# B&R Automation Studio project TD52 (part 146)

#### Stat_Obj.st - Cyclic code
```iecst
(*******************************************************************************
AGGR: read and write start statistic to windows file system	(cyclic)

This code is confidential and proprietary to the INNIO Company.
It may not be used in any form, or reproduced in any manner, without the express
written permission of the INNIO Company.
Copyright, INNIO Company, 2025

Customized modifications: -
------------------------

History:
-------
V4.06.00 	13-03-2018 	502423184	generated out of Stat_File
V4.06.01	20-07-2018	502423184	Erweitert um: LastRunInfo, TiAuxRel, Update(skip data info)
V4.12.00	29-03-2023	Kafka,		CBM HMI Handshake for Statistic Files
V4.13.0		30-10-2023	Kafka,		solve special sign issue
V4.14.0		27-02-2025	Perktold	added Ti_Purge_Dur to start statistic (new strVersion 4.14.0)

Instructions for use:
--------------------
Update Version number in the INIT program part and in history above!
Always increase the Version Number +0.00.01, if changes are made.

100ms+ Task class (TC6)

Outstandings:
------------
*******************************************************************************)

PROGRAM _INIT
(** A: Version Number *)
	strVersion			:=	'4.14.00';				(* Always increase the Version Number +0.00.01, if changes are made. *)

(** B: Initialize variables *)
	bOK 			:=	FALSE;
	aData			:=	ADR(szData);
	aTemp			:=	ADR(strTemp);
	lines			:=	1;
	strcpy(ADR(ModulName),ADR('CBM::Statistic'));

	pm_len			:=	SIZEOF(DerString_Stat);		(* define data length of permenent memory				*)

	DatObjInfo_01.enable		:=	TRUE;
	DatObjInfo_01.pName			:=	ADR(ModulName);

	DatObjCreate_01.enable		:=	TRUE;			(* enable create permanent memory data module FUB 		*)
	DatObjCreate_01.grp			:=	0;				(* must to be set to zero                  				*)
	DatObjCreate_01.pName		:=	ADR(ModulName);	(* set permanent memory data module name             	*)
	DatObjCreate_01.len			:=	pm_len;			(* set length of permanent memory data module         	*)
	DatObjCreate_01.MemType		:=	doUSRROM;		(* create permanent memory data module at USERROM   	*)
	DatObjCreate_01.Option		:=	0;				(* cyclic checksum monitoring is on            			*)
	DatObjCreate_01.pCpyData	:=	0;				(* no data will be copied do the perm. mem. data module	*)

	DatObjWrite_01.enable		:=	TRUE;			(* enable permanent memory data module read FUB 		*)
	DatObjWrite_01.Offset		:=	0;				(* start at memory offest zero                  		*)
	DatObjWrite_01.pSource		:=	ADR(DerString_Stat);	(* set permanent memory data module name		*)
	DatObjWrite_01.len			:=	pm_len;			(* set length ofpermanent memory data module        	*)

(** C: Functionality test and validation *)
	TON_Test.PT		:=	T#1m;
	bTest_Ena		:=	FALSE;

END_PROGRAM

PROGRAM _CYCLIC

(** 0: Functionality test and validation *)
	IF bTest_Ena THEN
		TON_Test.IN := NOT TON_Test.Q;
		TON_Test();

		IF TON_Test.Q THEN
			bStat_Write := TRUE;
			test_cnt	:=	(1 + test_cnt) MOD 3;
			iStat_Mode	:=	1 + test_cnt;
			CASE iStat_Mode OF
				1,2: 	lines			:=	StatSize;
				3:		lines			:=	Err.Size;
			END_CASE
		END_IF
	END_IF

(** 1: Triggers *)

(** 1.1: Statistic Triggers: manual trigger / automatic trigger every 100 starts *)
	IF iStep = _IDLE THEN
		IF VIS2MM.Stat.bTrig THEN
			bStat_Write		:=	TRUE;
			iStat_Mode		:=	MAN;
			lines			:=	StatSize;
		END_IF
		IF bStat_Trigger THEN
			bStat_Write		:=	TRUE;
			iStat_Mode		:=	AUTO;
			lines			:=	StatSize;
		END_IF
		VIS2MM.Stat.bTrig	:=	FALSE;
		bStat_Trigger		:=	FALSE;
	END_IF

(** 1.2: daily trigger for error counter myPlant *)
	IF NOT IN_CB.tPB2MM.bParaSetupOk THEN
		day_old			:=	tRealTime.day;
	END_IF
	IF tRealTime.day <> day_old THEN
		day_old			:=	tRealTime.day;
		bDaily_Trigger	:=	Para.iDailyTrigger_Ena > 0;
	END_IF

(** 1.3: Error Counter Trigger *)
	IF Para.bSA_PBC_Active AND iStep = _IDLE THEN
		IF VIS2MM.ErrCnt.bTrig OR bDaily_Trigger THEN
			bStat_Write		:=	TRUE;
			iStat_Mode		:=	ERRCNT;
			lines			:=	Err.Size;
		END_IF
		VIS2MM.ErrCnt.bTrig	:=	FALSE;
		bDaily_Trigger		:=	FALSE;
	END_IF

(** 2: initialiate file write *)
IF EDGEPOS(bStat_Write) THEN
	iStep 		:=	_BEGIN;
	bWrite		:=	TRUE;
	iZeile		:=	0;
	iOffset		:=	0;
	strFile			:=	'';																			(* create filename *)
	WRITE_Date(ADR(strFile),tRealTime);																(* Date *)
	IF iStat_Mode = ERRCNT THEN		strcat(ADR(strFile), ADR('_ErrCnt'));							(* _Name *)
	ELSE							strcat(ADR(strFile), ADR('_Statistic'));	END_IF
	strcat(ADR(strFile), ADR('_'));	strcat(ADR(strFile), ADR(IN_CB.szOrderID));						(* _OrderID *)
	strcat(ADR(strFile), ADR('_'));	itoa(IN_CB.iEngID, 	 aTemp);	strcat(ADR(strFile), aTemp);	(* _EngineID *)
	IF iStat_Mode = AUTO THEN		strcat(ADR(strFile), ADR('_Auto'));								(* _Mode *)
	ELSIF iStat_Mode = MAN THEN		strcat(ADR(strFile), ADR('_Man'));			END_IF
	strcat(ADR(strFile), ADR('.csv'));																(* .csv *)
END_IF

(** 3: when write process is done then reset event bit *)
	IF EDGENEG(bWrite) THEN
		bStat_Write	:=	FALSE;
	END_IF

(** 4: State machine *)
	CASE iStep OF
(** 4.1: write filename and version *)
	_BEGIN:
		szData		:=	'';
		strcat(aData, ADR('<STATS_NAME>'));																						(* ------------ *)
		strcat(aData, ADR(strFile));																							(* file name *)
		strcat(aData, ADR('</STATS_NAME><STATS_FILE>'));																		(* ------------ *)
		strcat(aData, ADR(strGEProp));																							(* GE prop info *)
		strcat(aData, ADR(strLine));																							(* ------------ *)
		strcat(aData, ADR('File_Version;'));	WRITE_STRING(ADR(strVersion),aData);				strcat(aData, ADR('$n'));	(* File version *)
		strcat(aData, ADR('Creation_Date;'));	WRITE_TS(tTimeStamp, aData);						strcat(aData, ADR('$n'));	(* Date & Time *)
		strcat(aData, ADR('J_Number;'));		WRITE_STRING(ADR(IN_CB.szOrderID),aData);			strcat(aData, ADR('$n'));	(* J Number *)
		strcat(aData, ADR('Motor_Number;'));	WRITE_DINT(IN_CB.iEngID,aData);						strcat(aData, ADR('$n'));	(* Serial ID *)
		strcat(aData, ADR('Engine_Type;'));		WRITE_DINT(xEngType.Motortype,aData);				strcat(aData, ADR('$n'));	(* Engine Type *)
		strcat(aData, ADR('Engine_Version;'));	WRITE_STRING(ADR(IN_CB.szEng_Motorversion),aData);	strcat(aData, ADR('$n'));	(* Engine Version *)
		strcat(aData, ADR('Trigger_Event;'));	WRITE_DINT(iStat_Mode,aData);						strcat(aData, ADR('$n'));	(* Trigger *)
		strcat(aData, ADR(strLine));																							(* ------------ *)

		DerString_Stat := '';
		iStrSize	:=	SIZEOF(DerString_Stat);
		iPointer	:=	ADR(DerString_Stat);
		iPointer	:=	save_strcat(ADR(DerString_Stat), iStrSize, iPointer, aData);					(* write data line *)
		iStep		:=	_HEAD;																			(* next step *)

(** 4.2: write file header *)
	_HEAD:
		szData		:=	'';
		IF iStat_Mode = AUTO OR iStat_Mode = MAN THEN													(* Statistic Header *)
			FOR i:=0 TO Stat.iSize DO	IF NOT Stat.i[i].Skip THEN	WRITE_STRING(ADR(Stat.i[i].Name), aData);	END_IF	END_FOR	(* Integer Names *)
			FOR i:=0 TO Stat.sSize DO	IF NOT Stat.s[i].Skip THEN	WRITE_STRING(ADR(Stat.s[i].Name), aData);	END_IF	END_FOR	(* String Names *)
			FOR i:=0 TO Stat.bSize DO	IF NOT Stat.b[i].Skip THEN	WRITE_STRING(ADR(Stat.b[i].Name), aData);	END_IF	END_FOR	(* Boolean Names *)
			FOR i:=0 TO Stat.rSize DO	IF NOT Stat.r[i].Skip THEN	WRITE_STRING(ADR(Stat.r[i].Name), aData);	END_IF	END_FOR	(* Real Names *)
			strcat(aData, ADR('$n'));
			FOR i:=0 TO Stat.iSize DO	IF NOT Stat.i[i].Skip THEN	WRITE_STRING(ADR(Stat.i[i].Unit), aData);	END_IF	END_FOR	(* Integer Units *)
			FOR i:=0 TO Stat.sSize DO	IF NOT Stat.s[i].Skip THEN	strcat(aData, ADR(';'));					END_IF	END_FOR	(* no Units *)
			FOR i:=0 TO Stat.bSize DO	IF NOT Stat.b[i].Skip THEN	strcat(aData, ADR(';'));					END_IF	END_FOR	(* no Units *)
			FOR i:=0 TO Stat.rSize DO	IF NOT Stat.r[i].Skip THEN	WRITE_STRING(ADR(Stat.r[i].Unit), aData);	END_IF	END_FOR	(* Real Units *)
			strcat(aData, ADR('$n'));
		ELSIF iStat_Mode = ERRCNT THEN																	(* ErrCounter Header *)
			strcat(aData, ADR('Reset date; '));			WRITE_TS(Err.tTS_Reset, aData);
			strcat(aData, ADR('$nReset OpHours; '));	itoa(Err.iCnt_OH_Reset,aTemp);	strcat(aData, aTemp);
			strcat(aData, ADR('$nWrite date; '));		WRITE_TS(tTimeStamp, aData);
			strcat(aData, ADR('$nWrite OpHours; '));	itoa(IN_CB.iCnt_OpHours,aTemp);	strcat(aData, aTemp);
			strcat(aData, ADR('$nErrorBit / Measurement; '));
			strcat(aData, ADR('Cyl / SAFI; '));
			strcat(aData, ADR('Counter; '));
			strcat(aData, ADR('First date; '));
			strcat(aData, ADR('Last date; '));
			strcat(aData, ADR('$n'));
		END_IF
		iPointer	:=	save_strcat(ADR(DerString_Stat), iStrSize, iPointer, aData);					(* write data line *)
		iStep		:=	_DATA;																			(* next step *)

(** 4.3: create data lines *)
	_DATA:
		szData		:=	'';																				(* clear previous data *)
		IF iStat_Mode = AUTO OR iStat_Mode = MAN THEN													(* Statistic Data *)
			iIdx	:=	(USINT_TO_INT(Stat.iIdx) - UDINT_TO_INT(iZeile) + USINT_TO_INT(StatSize + 1))MOD (StatSize + 1); (* calculate ring buffer index *)
			FOR i:=0 TO Stat.iSize DO	IF NOT Stat.i[i].Skip THEN	WRITE_DINT(Stat.i[i].Data[iIdx], 					aData);	END_IF	END_FOR
			FOR i:=0 TO Stat.sSize DO	IF NOT Stat.s[i].Skip THEN	WRITE_STRING(ADR(Stat.s[i].Data[iIdx].str), 		aData);	END_IF	END_FOR
			FOR i:=0 TO Stat.bSize DO	IF NOT Stat.b[i].Skip THEN	WRITE_BIT(Stat.b[i].Data[iIdx],						aData);	END_IF	END_FOR
			FOR i:=0 TO Stat.rSize DO	IF NOT Stat.r[i].Skip THEN	WRITE_REAL(Stat.r[i].Data[iIdx], Stat.r[i].Deci,	aData);	END_IF	END_FOR
		ELSIF iStat_Mode = ERRCNT THEN																	(* ErrCounter Data *)
			WRITE_STRING(ADR(ErrName[Err.xErr[iZeile].Name].str), 	aData);
			WRITE_DINT(Err.xErr[iZeile].iNum_Cyl, 					aData);
			WRITE_DINT(UDINT_TO_DINT(Err.xErr[iZeile].iCnt), 		aData);
			WRITE_TS(Err.xErr[iZeile].tTS_First,					aData);
			WRITE_TS(Err.xErr[iZeile].tTS_Last,						aData);
		END_IF
		strcat(aData, ADR('$n'));																		(* Line End *)
		iPointer	:=	save_strcat(ADR(DerString_Stat), iStrSize, iPointer, aData);					(* write data line *)
		IF iZeile < lines THEN			iZeile		:=	MIN(iZeile + 1, lines);							(* next line *)
		ELSE							iStep		:=	_FOOT;											(* next step *)
		END_IF

(** 4.4: create file footer *)
	_FOOT:
		iPointer	:=	save_strcat(ADR(DerString_Stat), iStrSize, iPointer, ADR('END OF FILE $n'));	(* last line *)
		iPointer	:=	save_strcat(ADR(DerString_Stat), iStrSize, iPointer, ADR('</STATS_FILE>'));		(* file end *)
		bWrite		:=	FALSE;																			(* write end *)
		iStep		:=	_EXIST;																			(* next step *)

(** 4.5: check for existing permanent memory data module *)
	_EXIST:
		DatObjInfo_01();
		CASE  DatObjInfo_01.status OF
		_BUSY: 	iStep;																					(* waiting *)
		_OKAY:	iStep 			:= _WRITE;																(* next step --> write the content to the flash disk	*)
				DatObjWrite_01.ident   	:= DatObjInfo_01.ident;											(* set identifier of permanent memory data module		*)
				DatObjWrite_01.len		:= pm_len;
		_DONF:	iStep		:=	_CREATE;																(* next step --> create permanent memory data module	*)
		ELSE	iErrorStep	:=	iStep;
				iStep		:=	_ERROR;
				iError		:=	DatObjInfo_01.status;
		END_CASE

(** 4.6: create permanent memory data module *)
	_CREATE:
		DatObjCreate_01();
		CASE  DatObjCreate_01.status OF
		_BUSY:	iStep;																					(* repeat until generation of permanent memory data module is ready *)
		_OKAY:	DatObjWrite_01.ident   	:= DatObjCreate_01.ident;										(* set identifier of permanent memory data module     	*)
				DatObjWrite_01.len		:= pm_len;
				iStep		:=	_WRITE;																	(* next step --> write the content to the flash disk	*)
		ELSE	iErrorStep	:=	iStep;
				iStep		:=	_ERROR;
				iError		:=	DatObjCreate_01.status;
		END_CASE

(** 4.7: write the content to the flash disk *)
	_WRITE:
		DatObjWrite_01();
	 	CASE DatObjWrite_01.status OF
		_BUSY:	iStep;																					(* repeat until write process of permanent memory data module is done *)
	   	_OKAY:	iStep				:=	_HMI;															(* next step --> wait for HMI to fetch file	*)
				xTON_HMI_Delay.IN	:=	TRUE;
		ELSE	iErrorStep			:=	iStep;
				iStep				:=	_ERROR;
				iError				:=	DatObjWrite_01.status;
		END_CASE

(** 4.8: wait FOR HMI TO fetch file	*)
	_HMI:
		MM2VIS.bStat_isCreated	:= TRUE;
		IF xTON_HMI_Delay.Q OR VIS2MM.bStat_isRead THEN
			iStep				:=	_DONE;																(* next step *)
			xTON_HMI_Delay.IN	:=	FALSE;
			MM2VIS.bStat_isCreated	:=	FALSE;
			VIS2MM.bStat_isRead		:=	FALSE;
		END_IF

(** 4.9: done, go to idle mode	*)
	_DONE:	iStep		:=	_IDLE;

(** 4.10: idle, reset lines	*)
	_IDLE:	iZeile		:=	0;
			iErrorStep	:=	0;

(** 4.11: error step, wait for cold start *)
	_ERROR: iStep;

(** 4.12: catch unexpected states *)
	ELSE	iErrorStep	:=	iStep;
			iStep		:=	_ERROR;
	END_CASE

(** 5: HMI Delay and out interfaces *)
	xTON_HMI_Delay.PT	:=	tiHMI_Delay;
	xTON_HMI_Delay();

	IF xTON_HMI_Delay.PT <> T#0s THEN
		rHMI_Delay	:=	LIMIT(0.0, TIME_TO_REAL(xTON_HMI_Delay.ET) / TIME_TO_REAL(xTON_HMI_Delay.PT), 1.0);
	ELSE
		rHMI_Delay	:=	0;
	END_IF

	IF iStep = _DONE THEN
		MM2VIS.Stat.rSave	:=	1.0;
	ELSIF iStep <> _HMI AND lines <> 0 THEN
		MM2VIS.Stat.rSave	:=	0.5 * UDINT_TO_REAL(iZeile)/UINT_TO_REAL(lines);
	ELSIF iStep = _HMI AND lines <> 0 THEN
		MM2VIS.Stat.rSave	:=	0.5 + 0.5 * rHMI_Delay;
	ELSIF iStep = _HMI AND lines = 0 THEN
		MM2VIS.Stat.rSave	:=	rHMI_Delay;
	END_IF

	MM2VIS.ErrCnt.rSave			:=	MM2VIS.Stat.rSave;

	MM2VIS.Stat.bSave			:=	iStep <> _IDLE AND lines = StatSize;
	MM2VIS.ErrCnt.bSave			:=	iStep <> _IDLE AND lines = Err.Size;

	IF iStep = _IDLE THEN
		MM2VIS.Stat.iStep			:=	USINT_TO_INT(_RDY);
		MM2VIS.ErrCnt.iStep			:=	USINT_TO_INT(_RDY);
	ELSE
		MM2VIS.Stat.iStep			:=	USINT_TO_INT(iStep) * BOOL_TO_INT(lines = StatSize) + _LOCK * BOOL_TO_INT(lines <> StatSize);
		MM2VIS.ErrCnt.iStep			:=	USINT_TO_INT(iStep) * BOOL_TO_INT(lines = Err.Size) + _LOCK * BOOL_TO_INT(lines <> Err.Size);
	END_IF

	MM2VIS.Stat.bLock			:=	iStep <> _IDLE;
	MM2VIS.ErrCnt.bLock			:=	iStep <> _IDLE;

END_PROGRAM
```

#### Stat_Obj.var - Local variables
```iecst
(********************************************************************
 * COPYRIGHT -- INNIO Company
 ********************************************************************
 * Program: PBC_MFile
 * File: PBC_MFile.var
 * Author: 502293141
 * Created: October 23, 2014
 ********************************************************************
 * Local variables of program PBC_MFile
 ********************************************************************)
VAR
	bOK : BOOL;
	strFile : STRING[50];
	iZeile : UDINT;
	iOffset : UDINT;
	iIdx : INT;
	bWrite : BOOL;
	szData : STRING[15000];
	iError : UINT;
	bStat_Write : BOOL;
	iStat_Mode : USINT;
	ModulName : STRING[32];
	pm_len : UDINT := 0;
	day_old : USINT;
	bDaily_Trigger : BOOL := 0;
	iStep : USINT := 0;
	DerString_Stat : STRING[200000];
	iErrorStep : INT;
	TON_Test : TON;
	i : UINT;
	strTemp : STRING[10];
	lines : UINT;
	DatObjCreate_01 : DatObjCreate;
	DatObjWrite_01 : DatObjWrite;
	DatObjInfo_01 : DatObjInfo;
	test_cnt : USINT;
	xTON_HMI_Delay : TON;
	strVersion : STRING[30];
	rHMI_Delay : REAL;
aData : UDINT;
aTemp : UDINT;
iStrSize : UDINT;
iPointer : UDINT;
END_VAR
VAR CONSTANT
	MAN : USINT := 1;
	AUTO : USINT := 2;
	ERRCNT : USINT := 3;
END_VAR
VAR
	bTest_Ena : BOOL := 0;
END_VAR
```

### Program Logical/CBM/Statistic/ErrCnt (IEC, version 4.06.1) - + counts errors

- ErrCnt.st (not readable text: treated as protected, skipped)

#### ErrCnt.var - Local variables
```iecst
(********************************************************************
 * COPYRIGHT -- INNIO Company
 ********************************************************************
 * Program: ErrCnt
 * File: ErrCnt.var
 * Author: 502423184
 * Created: December 14, 2015
 ********************************************************************
 * Local variables of program ErrCnt
 ********************************************************************)
VAR
	iNum_Cyl : USINT;
	iCnt : UINT;
	iCnt_Err : UINT;
	xTON_ErrCnt_Ena : TON;
END_VAR
VAR CONSTANT
	Knock_Int : USINT := 1;
	Knock_Lim : USINT := 2;
	Knock_Lim_Filt : USINT := 3;
	Misf_I : USINT := 4;
	Misf_II : USINT := 5;
	GlowIgn : USINT := 6;
	SensErr : USINT := 7;
	SensFailure : USINT := 8;
	MemBurst : USINT := 9;
	CPSSat : USINT := 0; (*Cylinder pressure sensor saturation - error counter*)
	CompLineCheck : USINT := 10;
	NegPresCheck : USINT := 11;
	PresSlopeCheck : USINT := 12;
	SlowDriftCheck : USINT := 13;
	PmaxLimReached : USINT := 14;
	NegVoltCheck : USINT := 15;
	ConfNotOK : USINT := 16;
	InvalidPar : USINT := 17;
	LimpHome : USINT := 18;
	OptiFreeze : USINT := 19;
END_VAR
```

### Program Logical/CBM/VisCBM (IEC) - Program

#### VisCBM.st - Cyclic code
```iecst
(*******************************************************************************
AGGR: VIS

This code is confidential AND proprietary to the INNIO Company.
It may NOT be used in any form, or reproduced in any manner, without the express
written permission of the INNIO Company.
Copyright, INNIO Company, 2019

Customized modifications: -
------------------------
History:
-------
V4.06.01 	30-07-2018 	502423184		header added, moved rCA_MFBxx to IN_CBM task

Instructions FOR use:
--------------------
- use in a 100ms cycle time

Outstandings:
------------
-

*******************************************************************************)
PROGRAM _INIT

	PINK;
END_PROGRAM

PROGRAM _CYCLIC

(** 1: colormap for that *)
	FOR i:= 1 TO 24 DO
		IF IN_CB.bTripCyl[i]				THEN	MM2VIS.iIdx_CylColor[i]	:=	RED;
		ELSIF IN_CB.bLimpHomeCylRKS_TC5[i]	THEN	MM2VIS.iIdx_CylColor[i]	:=	BLUE;
		ELSIF IN_CB.bLimpHomeCyl[i]			THEN	MM2VIS.iIdx_CylColor[i]	:=	YELLOW;
		ELSIF IN_CB.bSkipCylAct[i]			THEN	MM2VIS.iIdx_CylColor[i]	:=	GREY;
		ELSIF bATDCyl[i]					THEN	MM2VIS.iIdx_CylColor[i]	:=	VIOLET;
		ELSE 						 	 			MM2VIS.iIdx_CylColor[i]	:=	GREEN;
		END_IF
	END_FOR

(** 2: Statistic and CBM Screen visibility **)
	MM2VIS.bScreen_Stat :=	xEngType.Type9 OR Para.bSStat_Ena;
	MM2VIS.bScreen_CBM	:=	xEngType.Type9 OR Para.bSStat_Ena OR Para.bTCBMem_Ena OR Para.bECBMem_Ena OR Para.bSA_PBC_Active;

	MM2VIS.Stat.bScreen		:=	Para.bSStat_Ena;
	MM2VIS.ErrCnt.bScreen	:=	Para.bSA_PBC_Active;
	MM2VIS.TCB.bScreen		:=	Para.bTCBMem_Ena;
	MM2VIS.ECB.bScreen		:=	Para.bECBMem_Ena;

	MM2VIS.bFrictIMEP_Condition_On	:= OUT_CB.bFrictIMEP_Condition_On;

(** 3: SAFI data to HMI *)
	MM2VIS.rCA_MFB10 :=	rCA_MFB10;
	MM2VIS.rCA_MFB90 :=	rCA_MFB90;

END_PROGRAM
```

#### VisCBM.var - Local variables
```iecst
(********************************************************************
 * COPYRIGHT -- INNIO Company
 ********************************************************************
 * Program: VisCBM
 * File: VisCBM.var
 * Author: 105026853
 * Created: January 27, 2016
 ********************************************************************
 * Local variables of program VisCBM
 ********************************************************************)
VAR
	i : USINT;
END_VAR
```

### Program Logical/CBM/GnrlCBM (IEC) - Program

#### GnrlCBM.st - Cyclic code
```iecst
(*******************************************************************************
CBM: general monotioring task  (cyclic)

This code is confidential AND proprietary to the INNIO Company.
It may NOT be used in any form, or reproduced in any manner, without the express
written permission of the INNIO Company.
Copyright, INNIO Company, 2023

- GEN2diag checks the lambda movement AND shut down the engine in CASE OF a friciton event
- FricIMEP checks the friction power AND shut down the engine in CASE OF an increase

Customized modifications: -
------------------------

History:
-------

V4.05.0 xx-xx-2018 	Waldhart, 	created
V4.06.0 24-07-2018 	Waldhart, 	GEN2diag V0.3.9 implemented
		30-07-2018	502423184	replaced Para.bGEN2_preM_Act
V4.07.0 20-09-2018 	Waldhart, 	add containment for IMEP based friction monitoring rca
		09-10-2018 	Waldhart, 	IMEP based friction monitoring V0.06.0 implemented
		30-10-2018 	502423184, 	xGEN2diag von V4.6 übernommen
V4.09.0	23-01-2020	Schmidt,	GEN2diag: added interface for deactivation when LX2 is switched off
V4.10.0	22-07-2020	Schmidt,	IMEP based friction monitoring V0.07.1: exclude cylinders from monitoring if pressure sensor malfunction/error
V4.12.0	10-05-2022	Schmidt,	GEN2diag: increased delay for first activation to avoid FP detections while in GEN2 lambda minimum (issue #806)
V4.12.0	03-10-2022	Kafka,		desensitize voltage plausibility for IMEPbFricMon
		25-01-2023	Perktold, 	added variabel names to remove warnings after T9 task deactivation
V4.13.0	19-10-2023	Schmidt,	GEN2diag: for PBC deactivate monitoring during misfire (issue #1076)

Instructions FOR use:
--------------------

Outstandings:
------------

*******************************************************************************)
PROGRAM _INIT

	(*** GEN2 Friction monitoring ***)
	xGEN2diag.ssMethodType 		:= 3;

	(* transient detection *)
	xGEN2diag.Para.TrshPsetDev  		:= 0.02;	(* threshold value for power set point deviation [p.u.] *)
	xGEN2diag.Para.TrshPsetStat 		:= 0.02;	(* threshold value for steady state detection [p.u.] *)

	xGEN2diag.Para.TconstPsetStat 		:= 10.0;	(* timeconstant for steady state detection *)
	xGEN2diag.Para.TrshLoad 			:= 0.3;		(* threshold value for load level (related to the set power point) [p.u.] *)

	xGEN2diag.Para.TConstLP				:= 5.0; 	(* time constant [s] for the lambda lowpass filter *)
	xGEN2diag.Para.TConstHP             := 10.0; 	(* time constant [s] for the lambda highpass filter (situated after the lowpass) *)

	// TODO: type 4 0.014; type 3 0.01
	xGEN2diag.Para.ITPmeanScaling 		:= 0.014;	(* scaling for the mean ITP to estimate a lambda change *)

	xGEN2diag.Para.FaultThrshLambda     := 0.007; 	(* threshold value for lambda fault detection *)
	xGEN2diag.Para.TPulseLambdaFault    := 10.0; 	(* minimum time [s] a lambda fault pulse is provided for further detection (exh. temp.) *)
	xGEN2diag.Para.DeltaTexhAllowed     := 3.0; 	(* max. allowed rise in avg. exhaust temp. used for fault detection *)

	xGEN2diag.Para.TexhPlausibleMin 	:= 10;		(*min. exhaust temperature which is considered plausible (to exclude faulty sensors)*)
	xGEN2diag.Para.TexhPlausibleMax 	:= 850;		(*max. exhaust temperature which is considered plausible (to exclude faulty sensors)*)

	xGEN2diag.Para.WGM_FaultThrsh       := 0.1;     (*wastegate monitoring fault threshold*)
	xGEN2diag.Para.WGM_Tconst           := 1.0;     (*wastegate monitoring time constant*)

	xGEN2diag.Para.LEANOXErrorThrsh     := 0.01;   	(* threshold for leanox error (diagnosis gets active if the error is smaller than this threshold) *)
	xGEN2diag.Para.LEANOXErrorTconst	:= 1.0;		(*time constant [s] FOR filtering p2s in LEANOX error calculation'*)

	xGEN2diag.Para.Vltg_FaultThrsh      := 0.02;    (*voltage monitoring fault threshold*)
	xGEN2diag.Para.Vltg_Tconst          := 1;       (*voltage monitoring time constant*)

	xGEN2diag.Para.TexhSettledThrsh		:= 0.8;		(* threshold for exhaust temperature settled detection *)
	xGEN2diag.Para.TexhSettledTConstLP	:= 5;		(* time constant [s] for the Texh lowpass filter -> settled detection *)
	xGEN2diag.Para.TexhSettledTConstHP	:= 5;		(* time constant [s] for the Texh highpass filter (situated after the lowpass) -> settled detection *)
	xGEN2diag.Para.TexhSettledMaxTD		:= 15;		(* max. time [s] after a power ramp after which the exhaust temperature is considered settled (even if the filter does not suggest this! *)

	xGEN2diag.Para.bGasMixingEnDet		:= TRUE;	(* enable gas mixing threshold detection *)
	xGEN2diag.Para.GasMixingThrsh		:= 0.6;		(* threshold for gas mixing transient detection *)
	xGEN2diag.Para.GasMixingTconstLP	:= 5;		(* time constant [s] for gas mixing transient detection lowpass *)
	xGEN2diag.Para.GasMixingTconstHP	:= 5;		(* time constant [s] for gas mixing transient detection highpass *)

	(****************************************************************************************************************************)

	FricIMEP_P20.ssMethodType := 3;

	FricIMEP_P20.Para.PFComp_CC.Sig[0] := 1.0; 		FricIMEP_P20.Para.PFComp_CC.Comp[0] := 1.0;
	FricIMEP_P20.Para.PFComp_CC.Sig[1] := 0.9; 		FricIMEP_P20.Para.PFComp_CC.Comp[1] := 1.0;
	FricIMEP_P20.Para.PFComp_CC.Sig[2] := 0.8; 		FricIMEP_P20.Para.PFComp_CC.Comp[2] := 1.0;

	FricIMEP_P20.Para.PFComp_G_CC.Sig[0] := 0.25; 		FricIMEP_P20.Para.PFComp_G_CC.Comp[0] := 1.0;
	FricIMEP_P20.Para.PFComp_G_CC.Sig[1] := 0.63; 		FricIMEP_P20.Para.PFComp_G_CC.Comp[1] := 1.0;
	FricIMEP_P20.Para.PFComp_G_CC.Sig[2] := 1.0; 		FricIMEP_P20.Para.PFComp_G_CC.Comp[2] := 1.0;

	FricIMEP_P20.Para.WGComp_CC.WG_Pos[0] := 0.0; 		FricIMEP_P20.Para.WGComp_CC.Comp[0] := 1.0;
	FricIMEP_P20.Para.WGComp_CC.WG_Pos[1] := 0.5; 		FricIMEP_P20.Para.WGComp_CC.Comp[1] := 0.85;
	FricIMEP_P20.Para.WGComp_CC.WG_Pos[2] := 1.0; 		FricIMEP_P20.Para.WGComp_CC.Comp[2] := 0.7;

	FricIMEP_P20.Para.TEOComp_CC.TEO[0] := 40.0; 		FricIMEP_P20.Para.TEOComp_CC.Comp[0] := 1.3;
	FricIMEP_P20.Para.TEOComp_CC.TEO[1] := 80.0; 		FricIMEP_P20.Para.TEOComp_CC.Comp[1] := 1.0;
	FricIMEP_P20.Para.TEOComp_CC.TEO[2] := 120.0; 		FricIMEP_P20.Para.TEOComp_CC.Comp[2] := 1.0;

	FricIMEP_P20.Para.WGM_FaultThrsh	:= 0.02;	(* wastegate monitoring fault threshold*)
	FricIMEP_P20.Para.WGM_Tconst        := 1.0;     (* wastegate monitoring time constant*)
	FricIMEP_P20.Para.WGM_y0            := 0.0;     (* wastegate monitoring initial condition*)
	FricIMEP_P20.Para.WGM_TDly          := 5.0;     (* wastegate monitoring time delay*)

	FricIMEP_P20.Para.Vltg_FaultThrsh   := 200.0;	(* voltage monitoring fault threshold*)
	FricIMEP_P20.Para.Vltg_Tconst       :=   1.0;   (* voltage monitoring time constant*)
	FricIMEP_P20.Para.Vltg_y0           :=   0.0;   (* voltage monitoring initial condition*)
	FricIMEP_P20.Para.Vltg_TDly         :=   5.0;   (* voltage monitoring time delay [sec]*)

	FricIMEP_P20.Para.rTconst_Power_Filt := 4;		(* Time constant FOR Power filter *)
	FricIMEP_P20.Para.rTconst_fricflt_fastfilt := 4;(* Time constant OF friction power filter  - fast filtering *)
	FricIMEP_P20.Para.rTconst_fricflt_slowfilt := 8;(* Time constant OF friction power filter  - slow filtering *)
	FricIMEP_P20.Para.rIC_Power_filt := 0;

	FricIMEP_P20.Para.Abs_Thrsh 		:= 1132;	(* Threshold set TO compare the absolute value OF friction power FOR fault detection *)
	FricIMEP_P20.Para.Diff_Thrsh 		:= 36;		(* Threshold set TO compare the friction power difference value OF fast AND slow filter FOR fault detection *)

	FricIMEP_P20.Para.ExtDist_TDly      := 15.0;    (* time delay after a external disturbtion*)
	FricIMEP_P20.Para.rPower_Thrsh 		:= -500.0;	(* Power threshold TO switch on fault detection algorithm *)
	FricIMEP_P20.Para.Speedrange 		:= 5;		(* speed range [rpm] *)
	FricIMEP_P20.Para.rNEngNom 			:= 1000; 	(* nominal engine speed [rpm] *)
	FricIMEP_P20.Para.LoadStep_TDly 	:= 10;		(* time delay after a load step [sec] *)

	FricIMEP_P20.Para.rInertia 			:= 5460; 	(* inertia of engine plus generator [kgm2] *)
	FricIMEP_P20.Para.rEngine_Vd 		:= 0.0264;	(* Engine displacement volume *)

	FricIMEP_P20.Para.rD_P_kin 			:= 1; 		(* Derivative gain *)
	FricIMEP_P20.Para.rN_P_kin 			:= 5; 		(* Derivative filter *)
	FricIMEP_P20.Para.rD0_init 			:= 105; 	(*  *)
	FricIMEP_P20.Para.IMEPVali_Fac 		:= 8.0;		(* factor for the imep validation layer *)

	FricIMEP_P20.Para.rP_Nom			:= 9500;

(****************************************************************************************************************************)

(** just to remove compiler warnings after diabeling of type 9 tasks *)

	ACE2MM;
	FAM_ACN;
	FAM_pu_idx;
	FAM_status;
	FAM_value;
	FDT_Diag_1;
	FDT_Diag_10;
	FDT_Diag_11;
	FDT_Diag_12;
	FDT_Diag_13;
	FDT_Diag_14;
	FDT_Diag_15;
	FDT_Diag_16;
	FDT_Diag_17;
	FDT_Diag_18;
	FDT_Diag_19;
	FDT_Diag_2;
	FDT_Diag_20;
	FDT_Diag_21;
	FDT_Diag_22;
	FDT_Diag_23;
	FDT_Diag_24;
	FDT_Diag_25;
	FDT_Diag_26;
	FDT_Diag_27;
	FDT_Diag_28;
	FDT_Diag_29;
	FDT_Diag_3;
	FDT_Diag_30;
	FDT_Diag_31;
	FDT_Diag_32;
	FDT_Diag_33;
	FDT_Diag_34;
	FDT_Diag_35;
	FDT_Diag_36;
	FDT_Diag_37;
	FDT_Diag_38;
	FDT_Diag_39;
	FDT_Diag_4;
	FDT_Diag_40;
	FDT_Diag_41;
	FDT_Diag_42;
	FDT_Diag_43;
	FDT_Diag_44;
	FDT_Diag_45;
	FDT_Diag_46;
	FDT_Diag_47;
	FDT_Diag_48;
	FDT_Diag_49;
	FDT_Diag_5;
	FDT_Diag_50;
	FDT_Diag_51;
	FDT_Diag_52;
	FDT_Diag_53;
	FDT_Diag_54;
	FDT_Diag_55;
	FDT_Diag_56;
	FDT_Diag_57;
	FDT_Diag_58;
	FDT_Diag_59;
	FDT_Diag_6;
	FDT_Diag_60;
	FDT_Diag_7;
	FDT_Diag_8;
	FDT_Diag_9;
	Info_FAM;
	Info_FDT;
	MM2ACE;
	Version_FAM;
	Version_FDT;
	bFAM_CmdOn;
	bFDT_CmdOn;
	bGCB_ON_data;
	eta_gen;
	eta_mot;
	eta_vol;
	iCnt_OpHours;
	iOpHours_Min;
	rCosPhi_Max_data;
	rCosPhi_Min_data;
	rFrequency_Max_data;
	rFrequency_Min_data;
	rI_L1_Max_data;
	rI_L1_Min_data;
	rI_L2_Max_data;
	rI_L2_Min_data;
	rI_L3_Max_data;
	rI_L3_Min_data;
	rIgn_Timing_data;
	rLambda_Set_Max_data;
	rLambda_Set_Min_data;
	rMFBvar_data;
	rN_Eng_Max_data;
	rN_Eng_Min_data;
	rN_TCHP_A_Max_data;
	rN_TCHP_A_Min_data;
	rN_TCHP_B_Max_data;
	rN_TCHP_B_Min_data;
	rN_TCLP_A_Max_data;
	rN_TCLP_A_Min_data;
	rN_TCLP_B_Max_data;
	rN_TCLP_B_Min_data;
	rPI_Duration_data;
	rPI_Map_Offs_data;
	rPI_PID_Offs_data;
	rP_Act_Max_data;
	rP_Act_Min_data;
	rP_Set_Max_data;
	rP_Set_Min_data;
	rPos_CBV_Act_A1_Max_data;
	rPos_CBV_Act_A1_Min_data;
	rPos_CBV_Act_B1_Max_data;
	rPos_CBV_Act_B1_Min_data;
	rPos_CBV_Set_Max_data;
	rPos_CBV_Set_Min_data;
	rPr_49afTDC_data;
	rPr_49bfTDC_data;
	rPr_Crank_Case_Max_data;
	rPr_Crank_Case_Min_data;
	rPr_GR_Act_Max_data;
	rPr_GR_Act_Min_data;
	rPr_GR_Set_Max_data;
	rPr_GR_Set_Min_data;
	rPr_IMEP_data;
	rPr_Knock_data;
	rPr_Leanox_Set_Max_data;
	rPr_Leanox_Set_Min_data;
	rPr_P2s_A_Max_data;
	rPr_P2s_A_Min_data;
	rPr_P2s_B_Max_data;
	rPr_P2s_B_Min_data;
	rPr_PC_Act_Max_data;
	rPr_PC_Act_Min_data;
	rPr_PC_Set_Max_data;
	rPr_PC_Set_Min_data;
	rPr_Peak_data;
	rQ_Act_Max_data;
	rQ_Act_Min_data;
	rT_CBearing_data;
	rT_EG_Cyl_data;
	rT_MBearing_data;
	rT_T2s_data;
	rU_Ign_data;
	rU_L1L2_Max_data;
	rU_L1L2_Min_data;
	rU_L2L3_Max_data;
	rU_L2L3_Min_data;
	rU_L3L1_Max_data;
	rU_L3L1_Min_data;
	shiftVec;
	ulGlowIgn_data;
	ulLimpHome_data;
	ulMisfire_II_data;
	ulMisfire_I_data;
	ulPBCCompLineCheck_data;
	ulPBCMemBurst_data;
	ulPBCNegPresCheck_data;
	ulPBCNegVoltCheck_data;
	ulPBCPresSlopeCheck_data;
	ulPBCSensError_data;
	ulPBCSlowDriftCheck_data;
	ulSkipFire_data;

END_PROGRAM

PROGRAM _CYCLIC

	IF xEngType.Type6 THEN
		xGEN2diag.Para.TConstLP				:= 10.0; 	(* time constant [s] for the lambda lowpass filter *)
		xGEN2diag.Para.ITPmeanScaling 		:= 0.0228;	(* scaling for the mean ITP to estimate a lambda change *)
	ELSIF xEngType.Type4 THEN
		xGEN2diag.Para.TConstLP				:= 5.0; 	(* time constant [s] for the lambda lowpass filter *)
		xGEN2diag.Para.ITPmeanScaling 		:= 0.014;	(* scaling for the mean ITP to estimate a lambda change *)
	ELSIF xEngType.Type3 OR xEngType.Type2 THEN
		xGEN2diag.Para.TConstLP				:= 5.0; 	(* time constant [s] for the lambda lowpass filter *)
		xGEN2diag.Para.ITPmeanScaling 		:= 0.01;	(* scaling for the mean ITP to estimate a lambda change *)
	ELSE (*J920*)

	END_IF;

	xGEN2diag.Para.NCyl       			:= xEngType.NumberOfCylinder; 		(* number of cylinders *)
	xGEN2diag.Para.ThrshScale			:= Para.rScal_Lam_Mon_Limit;		(* GEN2 Scaling of Lambda monitoring Trip Threshold *)

	IF bGEN2diag_afterGCBon THEN
		xGEN2diag.Para.MonitoringDelay	:= 180.0;							(* GEN2 Lambda monitoring activation delay after engine start, increased delay to avoid false-positive detection by changing gas quality *)
	ELSE
		xGEN2diag.Para.MonitoringDelay	:= Para.rScal_Lam_Mon_Delay;		(* GEN2 Lambda monitoring activation delay *)
	END_IF;
	xGEN2diag.In.bFileOnlyInTrans		:= Para.bLam_Mon_ECBTCB_Ramps;		(* write files only (don't initiate a trip) during power ramps (only if detection is allowed during ramps) *)

	IF NOT xOpMode.NetP THEN
		bGEN2diag_afterGCBon := TRUE;
	ELSIF bLamMon_DiagActive THEN
		bGEN2diag_afterGCBon := FALSE;
	END_IF;

	xGEN2diag.In.bFileOnlyInTrans		:= Para.bLam_Mon_ECBTCB_Ramps;		(* write files only (don't initiate a trip) during power ramps (only if detection is allowed during ramps) *)

	(*** GEN2 Friction monitoring ***)
	xGEN2diag.In.bAllowDetInTrans 	:= Para.bLam_Mon_Act_Ramps; (*allow detection in transients*)

	xGEN2diag.In.Reset := NOT (xOpMode.NetP);

	xGEN2diag.In.bGasMixing_reset;
	xGEN2diag.In.rGasMixing_Ratio	:= IN_CB.rGT_RatioMix_TC2 * 100;

	xGEN2diag.In.Pset_norm			:= IN_CB.rP_Set_Norm; 		(*power reference trajectory [p.u.]*)
	xGEN2diag.In.Pset_WR_norm		:= IN_CB.rP_Set_GEN2_Norm; (* power reference without a ramp [p.u.]*)

	xGEN2diag.In.LambdaCmd 			:= IN_CB.rLam_Eng_LL_Set;

	xGEN2diag.In.p2s 				:= IN_CB.rPr_Ch_P2s_Avg_UF;	(*p2s [bar]*)
	xGEN2diag.In.p2sCmd 			:= IN_CB.rPr_Leanox_Set;	(*p2s command (LEANOX) [bar]*)

	xGEN2diag.In.posWG_norm 		:= IN_CB.rPos_Set_WG_Norm;	(*waste-gate position [p.u.] 0...1*)
	xGEN2diag.In.WGM_reset;							(*reset bit for the wastegate monitoring part*)

	xGEN2diag.In.LEANOXErrorFiltReset;				(*reset bit for the lowpass used to filter p2s in the LEANOX error settling detection*)

	xGEN2diag.In.bVltg_reset;						(*reset bit for the voltage monitoring part*)

	IF Para.rU_Gen_Nom[1] <> 0 THEN					(* nomalize the voltage *)
		xGEN2diag.In.U_L1L2_norm 		:= IN_CB.tU_L1L2[1].Ai / Para.rU_Gen_Nom[1];
		xGEN2diag.In.U_L2L3_norm 		:= IN_CB.tU_L2L3[1].Ai / Para.rU_Gen_Nom[1];
		xGEN2diag.In.U_L3L1_norm 		:= IN_CB.tU_L3L1[1].Ai / Para.rU_Gen_Nom[1];
	END_IF

	xGEN2diag.In.bGCBON 			:= IN_CB.tGCB_On.Di;
	xGEN2diag.In.bMCBON 			:= IN_CB.tMCB_On.Di;

	FOR i := 1 TO xEngType.NumberOfCylinder DO
		xGEN2diag.In.Texh[i-1] 		:= IN_CB.rT_EG_Cyl[i];		(* exhaust temperatures *)
	END_FOR

	xGEN2diag.In.Lambda_ss			:= IN_CB.rLamSteadyState;

	xGEN2diag.In.bTexhSettled_reset; 						(* reset bit for Texh settled detection (after power ramps) *)
	xGEN2diag.In.rITPmean := IN_CB.rCA_IgnP_Avg;			(* mean ignition timing point [°CA] *)

	(* monitor the inputs (leanox, Gride event and prechamber gas compressor *)

	(* check for parameter changes *)
	pm_len := SIZEOF(rDmyContainer);	(* measure the length to calulate the for loop *) (* 84 Byte // 21 Real PV´s *)
	ulChecksum := 0;					(* reset each time *)

	FOR iLoop := 0 TO 12 DO	(* loop over each datapackage *)

		ulOffset := 0;		(* reset of the offset *)

		CASE iLoop OF 		(* handle the worksplit *)

			1: 	memcpy(ADR(rDmyContainer) + ulOffset, ADR(Para.mp_a), SIZEOF(Para.mp_a)); ulOffset := ulOffset + SIZEOF(Para.mp_a);		(* 50 Bytes *)

			3: 	memcpy(ADR(rDmyContainer) + ulOffset, ADR(Para.mp_b), SIZEOF(Para.mp_b)); ulOffset := ulOffset + SIZEOF(Para.mp_b);		(* 50 Bytes *)

			5: 	memcpy(ADR(rDmyContainer) + ulOffset, ADR(Para.rCA_Ign_OP_Start), SIZEOF(Para.rCA_Ign_OP_Start)); ulOffset := ulOffset + SIZEOF(Para.rCA_Ign_OP_Start);		(* 20 Bytes *)
			 	memcpy(ADR(rDmyContainer) + ulOffset, ADR(Para.rCA_Ign_OP_Power), SIZEOF(Para.rCA_Ign_OP_Power)); ulOffset := ulOffset + SIZEOF(Para.rCA_Ign_OP_Power);		(* 20 Bytes *)
			 	memcpy(ADR(rDmyContainer) + ulOffset, ADR(Para.rCA_Ign_OP_Speed), SIZEOF(Para.rCA_Ign_OP_Speed)); ulOffset := ulOffset + SIZEOF(Para.rCA_Ign_OP_Speed);		(* 20 Bytes *)

			7:  memcpy(ADR(rDmyContainer) + ulOffset, ADR(Para.tLeanox_Comp_IgnP), SIZEOF(Para.tLeanox_Comp_IgnP)); ulOffset := ulOffset + SIZEOF(Para.tLeanox_Comp_IgnP);		(* 16 Bytes *)
				memcpy(ADR(rDmyContainer) + ulOffset, ADR(Para.bZZPKorr), SIZEOF(Para.bZZPKorr)); ulOffset := ulOffset + SIZEOF(Para.bZZPKorr);				(* 1 Bytes *)
				memcpy(ADR(rDmyContainer) + ulOffset, ADR(Para.bt2Korr), SIZEOF(Para.bt2Korr)); ulOffset := ulOffset + SIZEOF(Para.bt2Korr);				(* 1 Bytes *)
				memcpy(ADR(rDmyContainer) + ulOffset, ADR(Para.bDrehzkorr), SIZEOF(Para.bDrehzkorr)); ulOffset := ulOffset + SIZEOF(Para.bDrehzkorr);		(* 1 Bytes *)
				memcpy(ADR(rDmyContainer) + ulOffset, ADR(Para.tLeanox_Comp_ChTmp), SIZEOF(Para.tLeanox_Comp_ChTmp)); ulOffset := ulOffset + SIZEOF(Para.tLeanox_Comp_ChTmp);		(* 16 Bytes *)
				memcpy(ADR(rDmyContainer) + ulOffset, ADR(Para.rP_Eng_Frict), SIZEOF(Para.rP_Eng_Frict)); ulOffset := ulOffset + SIZEOF(Para.rP_Eng_Frict);			(* 4 Bytes *)
				memcpy(ADR(rDmyContainer) + ulOffset, ADR(Para.rP_Nom_Gastype), SIZEOF(Para.rP_Nom_Gastype)); ulOffset := ulOffset + SIZEOF(Para.rP_Nom_Gastype);	(* 20 Bytes *) (* 59 *)

			9:	memcpy(ADR(rDmyContainer) + ulOffset, ADR(Para.usHu), SIZEOF(Para.usHu)); ulOffset := ulOffset + SIZEOF(Para.usHu);		(* 20 Bytes *)
				memcpy(ADR(rDmyContainer) + ulOffset, ADR(Para.rMin_Air_Ratio), SIZEOF(Para.rMin_Air_Ratio)); ulOffset := ulOffset + SIZEOF(Para.rMin_Air_Ratio);		(* 40 Bytes *)

			11:	memcpy(ADR(rDmyContainer) + ulOffset, ADR(Para.usGasDensN), SIZEOF(Para.usGasDensN)); ulOffset := ulOffset + SIZEOF(Para.usGasDensN);		(* 20 Bytes *)
				memcpy(ADR(rDmyContainer) + ulOffset, ADR(Para.rPr_P2s_Set_LX_0kW), SIZEOF(Para.rPr_P2s_Set_LX_0kW)); ulOffset := ulOffset + SIZEOF(Para.rPr_P2s_Set_LX_0kW);		(* 40 Bytes *)

			2,4,6,8,10,12:
					FOR ulPMPointer := ADR(rDmyContainer) TO (ADR(rDmyContainer) + pm_len - SIZEOF(ulChkValue)) DO						(* split the dummy data container and  *)
						memcpy(ADR(ulChkValue), ulPMPointer, SIZEOF(ulChkValue));														(* sum-up the values --> *)
						ulChecksum := ulChecksum + ulChkValue;																			(* due to the overflow the *)
					END_FOR;																											(* one-way function creats a unique result *)
		ELSE
			bParaChange := FALSE;				(* reset the first time *)
		END_CASE
	END_FOR

	IF ulChecksum <> ulChecksumOld THEN (* check for changes *)
		ulChecksumOld := ulChecksum;	(* log the new value *)
		bParaChange := TRUE;			(* trigger the external settle time *)
	END_IF

	(* Leanox Controller *)
	bLeanoxChange := EDGEPOS(IN_CB.bLeanox_Man) OR EDGENEG(IN_CB.bLeanox_Man);
	bLeanoxM_Tgl := NOT xGEN2diag.In.bExt_dist AND IN_CB.bLeanox_Man; 					(* toggle as long as the leanox controller stays in manual mode *)

	(* Grid event *)
	bGrCChange := EDGEPOS(IN_CB.bMsg2831) OR EDGENEG(IN_CB.bMsg2831);

	(* PI Optimizer *)
	bPIOptiChange := EDGEPOS(IN_CB.bPIOptiChange);

	(* monitoring pressure prechamber gas compressor *)
	bPCGCChange := EDGEPOS(IN_CB.tPr_PCG_GC_Dem.Do) OR EDGENEG(IN_CB.tPr_PCG_GC_Dem.Do);

	(* PBC Misfire I or Misfire II bit *)
	bMisf_LGM := FALSE;
	FOR i := 1 TO xEngType.NumberOfCylinder DO
		IF IN_CB.bMisf_I[i] OR IN_CB.bMisf_II[i] THEN
			bMisf_LGM := TRUE;
		END_IF;
	END_FOR
	xTOF_Misf_LGM(IN := bMisf_LGM, PT := tiMisf_LGM);

	(* Sum-up the monitoring bits *)
	xGEN2diag.In.bExt_dist := bGEN2diag_Ext_dist := bParaChange OR bGrCChange OR bLeanoxChange OR bLeanoxM_Tgl OR bPIOptiChange OR IN_CB.bZylAusfallTP OR bPCGCChange OR IN_CB.bLX2_LGM_block OR xTOF_Misf_LGM.Q;

	xGEN2diag();

	bLGM_Event := (xGEN2diag.Out.FrictionFault) AND IN_CB.bGen2_NetP_ena; (* disable the observer alarms during service mode *)

	// trigger writing a file ONLY when a fault is detected during a power ramp -> appendix *_LGM_Ramp
	bLGM_Event_Ramp := (xGEN2diag.Out.FrictionFaultInTransient) AND IN_CB.bGen2_NetP_ena; 	(* disable the observer alarms during service mode *)

	bLamMon_DiagActive := xGEN2diag.dbgOut.DiagActive AND IN_CB.bGen2_NetP_ena;				(* diagnosis activated *)

	(* hand over the data for HMI trending *)
	MM2VIS.bLam_Mon_DiagAct := bLamMon_DiagActive;
	MM2VIS.rLam_Mon_Grad   	:= xGEN2diag.dbgOut.Residual;
	MM2VIS.rLam_Mon_TexhMin := xGEN2diag.dbgOut.TexhMin;
	MM2VIS.rLam_Mon_TexhAvg := xGEN2diag.dbgOut.TexhAvg;

(****************************************************************************************************************************)

	IF Para.rN_EngNom < 950 THEN 	(* 60Hz *)
		FricIMEP_P20.Para.PMEP_CC.P2_IP[0]	:= 1.35934; 			FricIMEP_P20.Para.PMEP_CC.PMEP_IP[0] := -0.1897;
		FricIMEP_P20.Para.PMEP_CC.P2_IP[1]	:= 2.126215; 		FricIMEP_P20.Para.PMEP_CC.PMEP_IP[1] := 0.0345;
		FricIMEP_P20.Para.PMEP_CC.P2_IP[2]	:= 3.00711; 			FricIMEP_P20.Para.PMEP_CC.PMEP_IP[2] := 0.2162;
		FricIMEP_P20.Para.PMEP_CC.P2_IP[3]	:= 3.9498; 			FricIMEP_P20.Para.PMEP_CC.PMEP_IP[3] := 0.3596;
		FricIMEP_P20.Para.PMEP_CC.P2_IP[4]	:= 4.4309; 			FricIMEP_P20.Para.PMEP_CC.PMEP_IP[4] := 0.4318;
		FricIMEP_P20.Para.PMEP_CC.P2_IP[5]	:= 4.92023; 			FricIMEP_P20.Para.PMEP_CC.PMEP_IP[5] := 0.512;
		FricIMEP_P20.Para.PMEP_CC.P2_IP[6]	:= 5.41085; 			FricIMEP_P20.Para.PMEP_CC.PMEP_IP[6] := 0.5814;
		FricIMEP_P20.Para.PMEP_CC.P2_IP[7]	:= 5.417585; 		FricIMEP_P20.Para.PMEP_CC.PMEP_IP[7] := 0.5844;
		FricIMEP_P20.Para.PMEP_CC.P2_IP[8]	:= 5.418; 			FricIMEP_P20.Para.PMEP_CC.PMEP_IP[8] := 0.5845;
		FricIMEP_P20.Para.PMEP_CC.P2_IP[9]	:= 5.419; 			FricIMEP_P20.Para.PMEP_CC.PMEP_IP[9] := 0.5846;
	ELSE							(* 50Hz *)
		FricIMEP_P20.Para.PMEP_CC.P2_IP[0]	:= 1.31; 			FricIMEP_P20.Para.PMEP_CC.PMEP_IP[0] := -0.2316;
		FricIMEP_P20.Para.PMEP_CC.P2_IP[1]	:= 1.728569; 		FricIMEP_P20.Para.PMEP_CC.PMEP_IP[1] := -0.1229;
		FricIMEP_P20.Para.PMEP_CC.P2_IP[2]	:= 2.17; 			FricIMEP_P20.Para.PMEP_CC.PMEP_IP[2] := -0.0343;
		FricIMEP_P20.Para.PMEP_CC.P2_IP[3]	:= 2.631067; 		FricIMEP_P20.Para.PMEP_CC.PMEP_IP[3] := 0.0383;
		FricIMEP_P20.Para.PMEP_CC.P2_IP[4]	:= 3.1; 				FricIMEP_P20.Para.PMEP_CC.PMEP_IP[4] := 0.0992;
		FricIMEP_P20.Para.PMEP_CC.P2_IP[5]	:= 3.590417; 		FricIMEP_P20.Para.PMEP_CC.PMEP_IP[5] := 0.1514;
		FricIMEP_P20.Para.PMEP_CC.P2_IP[6]	:= 4.08; 			FricIMEP_P20.Para.PMEP_CC.PMEP_IP[6] := 0.1943;
		FricIMEP_P20.Para.PMEP_CC.P2_IP[7]	:= 4.58; 			FricIMEP_P20.Para.PMEP_CC.PMEP_IP[7] := 0.2343;
		FricIMEP_P20.Para.PMEP_CC.P2_IP[8]	:= 5.09; 			FricIMEP_P20.Para.PMEP_CC.PMEP_IP[8] := 0.2815;
		FricIMEP_P20.Para.PMEP_CC.P2_IP[9]	:= 5.62; 			FricIMEP_P20.Para.PMEP_CC.PMEP_IP[9] := 0.3252;
	END_IF

	FricIMEP_P20.Para.NumberOfCylinder 		:= xEngType.NumberOfCylinder;		(* Engine no OF cylinders *)
	FricIMEP_P20.Para.rInertia 		  		:= Para.rGen_Inertia; 				(* inertia of engine plus generator [kgm2] *)
	FricIMEP_P20.Para.rP_Nom	 			:= IN_CB.rP_Nom;
	FricIMEP_P20.Para.rNEngNom				:= Para.rN_EngNom;

	FricIMEP_P20.In.Speed 					:= IN_CB.rN_IgnSAFI_Act;			(* engine speed *)
	FricIMEP_P20.In.Pact 					:= IN_CB.tP_Act[1].Unfilt;
	FricIMEP_P20.In.bGCBON 					:= IN_CB.tGCB_On.Di;
	FricIMEP_P20.In.bMCBON 					:= IN_CB.tMCB_On.Di;

	FricIMEP_P20.In.PF_Act  				:= IN_CB.tPF_Act[1].Ai;
	FricIMEP_P20.In.T_EO  					:= IN_CB.tT_EO.Ai;
	FricIMEP_P20.In.rPos_Set_WG_Norm;

	FricIMEP_P20.In.U_L1L2					:= IN_CB.tU_L1L2[1].Unfilt;
	FricIMEP_P20.In.U_L2L3					:= IN_CB.tU_L2L3[1].Unfilt;
	FricIMEP_P20.In.U_L3L1					:= IN_CB.tU_L3L1[1].Unfilt;

	FricIMEP_P20.In.I_L1					:= IN_CB.tI_L1[1].Unfilt;
	FricIMEP_P20.In.I_L2					:= IN_CB.tI_L2[1].Unfilt;
	FricIMEP_P20.In.I_L3					:= IN_CB.tI_L3[1].Unfilt;

	FricIMEP_P20.In.rPrChP2s  				:= IN_CB.rPr_Ch_P2s_Avg_UF;			(* unfiltered Average charge pressure p2' (after throttle valve) [bar] *)

	FricIMEP_P20.In.rPos_Set_WG_Norm		:= IN_CB.rPos_Set_WG_Norm; 			(* handover the setpoint for the waste gate position *)

	FricIMEP_P20.In.Reset_fastfilt := FricIMEP_P20.In.Reset_slowfilt := EDGEPOS(IN_CB.tGCB_On.Di) OR EDGENEG(IN_CB.tGCB_On.Di);

	FricIMEP_P20.In.bExt_dist := EDGEPOS(IN_CB.bMsg2831) OR EDGENEG(IN_CB.bMsg2831); 	(* Grid event *)

	FOR i := 1 TO xEngType.NumberOfCylinder DO
		FricIMEP_P20.In.bPBCSensErr[i] 		:= IN_CB.bPBCSensErr[i];
		FricIMEP_P20.In.rPrIMEP[i] 			:= IN_CB.rPr_IMEP[i];
		FricIMEP_P20.In.bLimpHomeCyl[i] 	:= IN_CB.bLimpHomeCyl[i];
		FricIMEP_P20.In.bLimpHomeCylG2[i] 	:= IN_CB.bLimpHomeCylRKS[i];
		FricIMEP_P20.In.bLimpHomeCylExt[i] 	:= FALSE;
	END_FOR

	(*** IMEP Monitoring ***)
	FricIMEP_P20();

	bFMEP_Fault_Detection := FricIMEP_P20.Out.Fault_Diff AND Para.bFMEP_enable AND NOT (bGnlTrip AND IN_CB.tP_Act[1].Ai < (IN_CB.rP_Nom * 0.4));	(* hand-over to the MsgCB task *)

	OUT_CB.bFrictIMEP_Condition_On := FricIMEP_P20.dbgOut.Condition_ON AND Para.bFMEP_enable;

(****************************************************************************************************************************)

END_PROGRAM
```

#### GnrlCBM.var - Local variables
```iecst
(********************************************************************
 * COPYRIGHT -- INNIO Company
 ********************************************************************
 * Program: GnrlCBM
 * File: GnrlCBM.var
 * Author: 105026853
 * Created: June 13, 2016
 ********************************************************************
 * Local variables of program GnrlCBM
 ********************************************************************)
VAR
	xGEN2diag : fGEN2diag := (0);
	bGrCChange : BOOL := 0;
	pm_len : UINT := 0;
	rDmyContainer : ARRAY[0..20] OF REAL;
	ulChecksum : UDINT := 0;
	iLoop : USINT := 0;
	ulOffset : UINT := 0;
	ulPMPointer : UDINT := 0;
	ulChkValue : UDINT := 0;
	bParaChange : BOOL := 0;
	ulChecksumOld : UDINT := 0;
	bLeanoxChange : BOOL := 0;
	bLeanoxM_Tgl : BOOL := 0;
	bPIOptiChange : BOOL := 0;
	i : USINT;
	FricIMEP_P20 : fFricIMEP := (0);
	bPCGCChange : BOOL := 0;
	bGEN2diag_afterGCBon : BOOL := 0;
	xTOF_Misf_LGM : TOF;
	tiMisf_LGM : TIME := T#60s;
	bMisf_LGM : BOOL;
END_VAR
```

### Program Logical/CBM/PermCBM (IEC) - Program

#### PermCBMCyclic.st - Cyclic code
```iecst
(*******************************************************************************
AGGR: read AND write DIA.NE XT parameter TO flash memory	(cyclic)

This code is confidential and proprietary to the INNIO Company.
It may not be used in any form, or reproduced in any manner, without the express
written permission of the INNIO Company.
Copyright, INNIO Company, 2019

- every 10 seconds or at write once the parameter values are copied to the structure pm
- every 10 seconds the checksum of the parameter structure is calculate
- if checksum has changed or write once is set the structure pm is written to
	the permanent memory data module

Customized modifications: -
------------------------

History:
---
-after successful prem write, all further write attempts will be delayed for 10min to reduce flash wear----
V04.09.00.00	28-05-2019	Waldhart,	generated
				10.09.2019	Zengerer	Basisupdate01 from V4.07 implemented: Changed Perm Storage Handling for reduced file write cycle -10min delay after successful prem write

 *
 * Customized modifications: -
 * ------------------------
 * This is the customized Version for METAMODULE CB
 *
 * Outstandings:
 * ------------
 *
 ********************************************************************)

(***********************************************************************************************************)
(* CYCLIC **************************************************************************************************)
(***********************************************************************************************************

Instructions FOR use:
--------------------
(* MODULE SPECIFIC CHANGES IN CYCLIC PART:
 * Confgure IN_CU and OUT_CU Structure names in cyclic task.
 * Configure optional checking for necessary Parameter in cyclic task.

(**********************************************************************************************************)

PROGRAM _CYCLIC

	(* participate in parasave environment to use system status messages: *)
	(* Connection from tParaIntern structure to IN and OUT structures INSTRUCTION: EDIT 1xIN_ and 2xOUT_ STRUCTURE NAMES FOR THIS MODULE HERE! *)
	tParaIntern.tParaBase2MM	:= IN_CB.tPB2MM;
	(*OUT_CB.tCB2PB.				:= tParaIntern.tMM2ParaBase.;  DO NOT CONNECT ParaOUT STRUCTURE HERE in Perm task! *)

(********************************************************************************************************)
(* Every 10 seconds OR at write once the parameter values are copied TO the 							*)
(* structure pm. Afterwards the structure pm is written TO the permanent memory							*)
(* module IF the checksum OF the parameter struct has been changed.										*)
(**********************************************************************************************************)
	(* 10 seconds timer *)
	TON_WritePMEM(IN := NOT TON_WritePMEM.Q, PT:= T#10s);
	TON_BlockMinFileAge(IN := bBlock_MinFileAge, PT:= T#10m);			(*V4.07.1 reduced Perm file write intervall*)
	IF TON_BlockMinFileAge.Q  THEN bBlock_MinFileAge := FALSE; END_IF	(*V4.07.1 reduced Perm file write intervall*)

	(* every 10 seconds or at write once the parameter values are copied to the structure pm *)
	IF TON_WritePMEM.Q OR write_once THEN

	(************ Permanent structure ************)
		pmm				:= Perm;

		pmm.iSpare_5	:= iPM_WriteCnt;		(*Perm diagnosis value implemented in V4.07.1; may be removed and used for other topics later on, if necessary *)

	END_IF;

	(* cyclic calcualtion of parameter checksum	*)
	IF TON_WritePMEM.Q THEN
		ulChecksum := 0;

		FOR ulPMPointer := ADR(pmm) TO (ADR(pmm) + pm_len - SIZEOF(ulChkValue)) DO
			memcpy(ADR(ulChkValue), ulPMPointer, SIZEOF(ulChkValue));
			ulChecksum := (ulChecksum XOR ulChkValue)+ulChkValue;
		END_FOR;

		IF ulChecksumOld <> ulChecksum THEN	(* if checksum has changed 		*)
			ulChecksumOld := ulChecksum;	(* save last cheksum value		*)
			bWriteDataObj := TRUE;			(* set flag for write checksum	*)
		END_IF;

	END_IF

	(* write structure pm to the permanent memory module  	changed with bBlock_MinFileAge V4.07.1, for reduced Perm file write intervall*)
	IF ( (bWriteDataObj AND NOT bBlock_MinFileAge) OR write_once ) AND tParaIntern.tParaBase2MM.bSaveParaAllowed AND NOT tParaIntern.tParaBase2MM.bDownloadDetected THEN

		DatObjWrite_01();									(* run data object write fub 				*)

		IF DatObjWrite_01.status <> ERR_FUB_BUSY THEN		(* wait if data object write fub is busy 	*)
			bWriteDataObj 	:= FALSE;						(* reset data object write flag				*)
			write_once 		:= FALSE;						(* reset write_once flag 					*)
			iPM_WriteCnt 	:= iPM_WriteCnt  + 1;			(* former usPMWriteCnt: counter for done data object module writes *)

			IF OUT_CB.tCB2PB.iPermStatus >=0 THEN 												(* new V4.06: if not already on error state, then transmit this perm status info *)
				OUT_CB.tCB2PB.iPermStatus := LIMIT(2, OUT_CB.tCB2PB.iPermStatus + 1, 999);		(* new V4.06: transmit OK= positive perm status info *)
				IF OUT_CB.tCB2PB.iPermStatus = 999 THEN OUT_CB.tCB2PB.iPermStatus := 2; END_IF	(* new V4.06: transmit OK= positive perm status info *)
				OUT_CB.tCB2PB.bPermSetupOk := TRUE	;											(* new V4.06: transmit perm status info *)
			END_IF

			IF DatObjWrite_01.status = ERR_NOERROR THEN		(* if error status NO ERROR, then start timer to block forther write requests for some time to avoid CF wear down	*)
				bBlock_MinFileAge := TRUE;
			ELSE											(* if error status not no error 			*)
				pm_Error := 1004;							(* set data object write error state		*)
			END_IF;
		END_IF;

	END_IF;

//OLD	(* set RPS warning if no access to SysRom file is possible *)
//OLD	TON_WarnDelay(IN := pm_Error > 3 OR NOT tParaIntern.tParaBase2MM.bSaveParaAllowed, PT:= T#15s);
//OLD	tParaIntern.tMM2ParaBase.bMyParaMissing	:= TON_WarnDelay.Q; 	(*replacement for RPSW[1] := *)

	(* Forward Perm Error - new V4.06 *)
//	IF (pm_Error > 0) AND (OUT_CB.tCB2PB.iPermStatus <= 0) THEN OUT_AG.tAG2PB.iPermStatus := LIMIT(-999999,-pm_Error ,-1) ;	END_IF		(*no CYCLIC! new V4.06: transmit error as negative perm status info *)
	IF (pm_Error > 0) AND (OUT_CB.tCB2PB.iPermStatus >= 0) THEN 	OUT_CB.tCB2PB.iPermStatus :=LIMIT(-999999,-UINT_TO_DINT(pm_Error) ,-1);	END_IF		(* new V4.06: transmit error as negative perm status info *)
	IF (OUT_CB.tCB2PB.iPermStatus < 0) THEN 	OUT_CB.tCB2PB.bPermSetupOk := FALSE	;	END_IF			(* new V4.06: transmit perm status info *)

END_PROGRAM

(***********************************************************************************************************)
PROGRAM _EXIT

	tParaIntern.tMM2ParaBase.bMySys_Run := FALSE;				(* local 'RUN' and 'run_plc' clearing*)
	//REMOVED IF NOT bOpt_PermDataWrite_Continuous THEN			(* alternative attempt to write perm file only on EXIT*)

END_PROGRAM
```

#### PermCBMInit.st - Initialization code
```iecst
(*******************************************************************************
AGGR: read AND write DIA.NE XT parameter TO flash memory	(init)

This code is confidential AND proprietary TO the INNIO Company.
It may NOT be used in any form, or reproduced in any manner, without the express
written permission OF the INNIO Company.
Copyright, INNIO Company, 2019

- every 10 seconds OR at write once the parameter values are copied TO the structure pm
- every 10 seconds the checksum OF the parameter structure is calculate
- IF checksum has changed OR write once is set the structure pm is written TO
	the permanent memory data module

Customized modifications: -
------------------------

History:
-------
V04.09.00.00	28-05-2019	Waldhart,	generated
				10.09.2019	Zengerer	Basisupdate01 from V4.07 implemented: Changed Perm Storage Handling for reduced file write cycle -10min delay after successful prem write

Instructions FOR use:
--------------------
(init)
The parameter are stored in a data module which is stored on flash memory.
At start up the parameter will be readed from the flash memory AND copied TO
the parameter variables. If the data module does NOT exist OR the length OF
data module AND parameter struct is different, the data module will be created.
(cyclic)
Every 10 seconds OR at write once the parameter values are copied TO the
structure pm. Afterwards the structure pm is written TO the permanent memory
module IF the checksum OF the parameter struct has been changed.

Add new tags only at the end OF the structure AND check/INSERT new data module lenght!

Outstandings:
------------
*******************************************************************************)

PROGRAM _INIT

	(* set some init parameters *)
	TON_WritePMEM(IN := FALSE, PT:= T#10s);			(* reset used timer function blocks 			*)

	pm_Error 	:= ERR_NOERROR;						(* reset permanent memory error	status			*)
	write_once 	:= FALSE;				 			(* reset flag for write permanent memory once	*)
	pm_len 		:= SIZEOF(pmm);						(* define data length of permenent memory		*)
	strcpy(ADR(ModuleName),ADR('CBM::CBM_perm'));			(* define name of permanent memory data module	*)

	(* check for existing permanent memory data module	*)
	DatObjInfo_01.enable:= TRUE;					(* enable FUB									*)
	DatObjInfo_01.pName := ADR(ModuleName);			(* set permanent memory data module name 		*)
	DatObjInfo_01();								(* run data object info FUB						*)

	(* check error status of data object info FUB	*)
	IF DatObjInfo_01.status = ERR_NOERROR THEN		(* if no error	--> permanent memory data module exists	*)
		pm_id 	:= DatObjInfo_01.ident;				(* copy permanent memory data module ident			*)
		pm_p 	:= DatObjInfo_01.pDatObjMem;		(* copy permanent memory data module memory adres	*)
	ELSE
		bCreateDataObj := TRUE;						(* set flag for create new data object	*)
		pm_Error := 1001;							(* set permanent memory error status	*)
	END_IF;

	(* check length of parameter struct with length of data object *)

	IF DatObjInfo_01.len = pm_len THEN
			perm_par_vers  := 409;			(* 409 = length of perm_par V4.09.0 *) //update FS structure

	ELSE
			bCreateDataObj := TRUE;			(* set flag for create new data object	*)
	END_IF

	(* if permanent memory data module exist read data and copy to structure pm	*)
	IF pm_Error = ERR_NOERROR THEN					(* permanent memory data module exist 				*)
		DatObjRead_01.enable 		:= TRUE;		(* enable read permanent memory module data 		*)
		DatObjRead_01.ident 		:= pm_id;		(* set identifier of permanent memory data module	*)
		DatObjRead_01.Offset 		:= 0;			(* start at memory offest zero 						*)
		DatObjRead_01.pDestination := ADR(pmm);		(* set permanent data destination adress			*)
		DatObjRead_01.len 			:= DatObjInfo_01.len;	(* set length of permanent data module		*)

		REPEAT	(* repeat until data of permanent memory data module have been read *)
			DatObjRead_01();						(* FUB read data from permanent data module 		*)
			UNTIL	DatObjRead_01.status <> ERR_FUB_BUSY		(* wait if FUB is busy 	*)
		END_REPEAT;

		IF DatObjRead_01.status <> ERR_NOERROR THEN	(* if status of read permanent data moduel is not OK 	*)
			pm_Error := 1002;						(* set permanent memory error status					*)
		ELSE
			IF OUT_CB.tCB2PB.iPermStatus >=0 THEN 													(* new V4.06: transmit perm status info *)
				OUT_CB.tCB2PB.iPermStatus := LIMIT(2, OUT_CB.tCB2PB.iPermStatus + pm_len, 999999);	(* new V4.06: transmit perm status info *)
				OUT_CB.tCB2PB.bPermSetupOk := TRUE	;												(* new V4.06: transmit perm status info *)
			END_IF																					(* new V4.06: transmit perm status info *)
		END_IF
	END_IF

	(* if permanent memory data module exist --> copy data from structure pm to program parameter *)
	IF pm_Error = ERR_NOERROR THEN

		(*************************)
		Perm						:= pmm;				(* overall copy of values from stored structure 'pm' to active structure 'Perm'  *)

		iPM_WriteCnt				:= pmm.iSpare_5;	(* Perm diagnosis value implemented in V4.07.1; may be removed and used for other topics later on, if necessary*)

		   IF OUT_CB.tCB2PB.iPermStatus >=0 THEN 												(* new V4.06: transmit perm status info *)
				OUT_CB.tCB2PB.iPermStatus := LIMIT(2, OUT_CB.tCB2PB.iPermStatus + pm_len, 999);	(* new V4.06: transmit perm status info *)
		   		OUT_CB.tCB2PB.bPermSetupOk := TRUE	;											(* new V4.06: transmit perm status info *)
			END_IF																				(* new V4.06: transmit perm status info *)

		(*************************)

	END_IF;

	(* create new permanent memory data module	*)
	IF bCreateDataObj THEN

//		(* try to delete old data module *)
//		DatObjDelete_PermMem.enable := TRUE;		(*OLD! NOT POSSIBLE IN SYSROM! *)

		(* create new one *)
		DatObjCreate_01.enable	 := TRUE;			(* enable create permanent memory data module FUB 	*)
		DatObjCreate_01.grp 	 := 0;				(* must to be set to zero							*)
		DatObjCreate_01.pName 	 := ADR(ModuleName);	(* set permanent memory data module name 			*)
		DatObjCreate_01.len 	 := pm_len;			(* set length ofpermanent memory data module		*)
		DatObjCreate_01.MemType  := doUSRROM;		(* create permanent memory data module at USERROM (changed from doSYSROM due to VIS reasons)	*)
		DatObjCreate_01.Option 	 := 0;				(* cyclic checksum monitoring is on					*)
		DatObjCreate_01.pCpyData := 0;				(* no data will be copied do the permanent memory data module *)

		pm_Error:= 1003;							(* set permanent memory error status	*)

		REPEAT	(* repeat until generation of permanent memory data module is ready *)
			DatObjCreate_01();						(* FUB for create permanent memory data module 		*)
			UNTIL	DatObjCreate_01.status <> ERR_FUB_BUSY		(* wait if FUB is busy 	*)
		END_REPEAT;

		IF DatObjCreate_01.status = ERR_NOERROR THEN	(* is creation of permanent memory data module OK 	*)
			pm_p 	:= DatObjCreate_01.pDatObjMem;		(* set memory adress of permanent memory data module*)
			pm_id 	:= DatObjCreate_01.ident;			(* set identifier of permanent memory data module 	*)
		ELSE
			pm_Error:= 1004;							(* set permanent memory error status	*)
		END_IF;
	END_IF;

	(* prepare parameter for permanent memory data write in cyclic task *)
	IF pm_Error < 4 THEN							(* permanent memory data module exist or has been created	*)
		DatObjWrite_01.enable 	:= TRUE;			(* enable permanent memory data module read FUB 	*)
		DatObjWrite_01.ident 	:= pm_id;			(* set identifier of permanent memory data module 	*)
		DatObjWrite_01.Offset 	:= 0;				(* start at memory offest zero 						*)
		DatObjWrite_01.pSource 	:= ADR(pmm);		(* set permanent memory data module name 			*)
		DatObjWrite_01.len 		:= pm_len;			(* set length ofpermanent memory data module		*)
	END_IF;

	(* calcualte actual checksum of parameter structure	*)
	ulChecksumOld := 0;			(* reset checksum value *)

	FOR ulPMPointer := ADR(pmm) TO (ADR(pmm) + pm_len - SIZEOF(ulChkValue)) DO
		memcpy(ADR(ulChkValue), ulPMPointer, SIZEOF(ulChkValue));
		ulChecksumOld := ulChecksumOld XOR ulChkValue;
	END_FOR;

	(**Forward Perm Error - new V4.06 *)
	IF (pm_Error > 0) AND (OUT_CB.tCB2PB.iPermStatus = 0) THEN 	OUT_CB.tCB2PB.iPermStatus := - pm_Error	;	END_IF		(* new V4.06: transmit error as negative perm status info *)
	IF (OUT_CB.tCB2PB.iPermStatus < 0) THEN 	OUT_CB.tCB2PB.bPermSetupOk := FALSE	;	END_IF			(* new V4.06: transmit perm status info *)

END_PROGRAM
```

#### PermCBM.var - Package variables
```iecst
VAR
	tParaIntern : ParaHandler_typ; (*Connector type to perm_par*)
	bWriteDataObj : BOOL; (* TRUE=write data object module *)
	bCreateDataObj : BOOL; (* TRUE=create new data object *)
	write_once : BOOL; (* write permanent memory once *)
	DatObjCreate_01 : DatObjCreate; (* data object create *)
	DatObjInfo_01 : DatObjInfo; (* data object info *)
	DatObjRead_01 : DatObjRead; (* data object read *)
	DatObjWrite_01 : DatObjWrite; (* data object write *)
	ModuleName : STRING[35]; (* module name of object *)
	TON_WritePMEM : TON; (* delay write permanent memory *)
	ulPMPointer : UDINT; (* adress of actual checksum value *)
	ulChecksum : UDINT; (* parameter checksum value *)
	pm_len : UDINT; (* permanent value lenght *)
	ulChecksumOld : UDINT; (* last vlaue of parameter checksum *)
	ulChkValue : UDINT; (* actual value of parameter pointer *)
	pm_id : UDINT; (* permanent value identifier *)
	pm_p : UDINT; (* permanent value pointer *)
	perm_par_vers : UINT;
END_VAR
VAR CONSTANT
	ERR_NOERROR : UINT := 0;
END_VAR
VAR
	pmm : Perm_CBM_Struct;
	pm_Error : UINT; (* permanent value error *) (* Deleted: pm : ParaMem_typ; permanent memory tags mathias, 22.8.11*)
	TON_BlockMinFileAge : TON; (*waiting time without file write after successful performed write*)
	bBlock_MinFileAge : BOOL := FALSE; (*pause the perm file write after each sucessful write*)
	iPM_WriteCnt : UDINT; (* *) (*old VarName: usPMWriteCnt*)
END_VAR
```

### Package Logical/DataInterface - DI: DataInterface for Testbench
